// TIA Portal project "lab1" (V15.1)

(* hardware
DEVICE "S7-1200 station_1"  S7-1200 Station
   slot 0: "Rack_0"  S7-1200 Rack  Rack  V1.0
   slot 1: "PLC_1"  CPU 1214C AC/DC/Rly  6ES7 214-1BG40-0XB0  V4.2
*)

// ===== PLC "PLC_1"  CPU 1214C AC/DC/Rly =====

VAR_GLOBAL   // PLC tag table "Default tag table"
   "START_NO" AT %I0.1 : Bool;
   "MOTOR_RADI_NO" AT %I0.2 : Bool;
   "AUTOMATSKI_REZIM_NO" AT %I0.3 : Bool;
   "STOP_NO" AT %I0.5 : Bool;
   "SAFETY_RELE_NC" AT %I0.6 : Bool;
   "ZASTITNI_PREKIDAC_NO" AT %I1.0 : Bool;
   "KONTAKTOR_UKLJUCEN_NO" AT %I1.1 : Bool;
   "ZELENI_LED" AT %Q0.0 : Bool;
   "CRVENI_LED" AT %Q0.1 : Bool;
   "KONTAKTOR_IZLAZ" AT %Q0.2 : Bool;
   "KVAR_ZASTITNI_PREKIDAC" AT %M0.0 : Bool;
   "KVAR_KONTAKTOR" AT %M0.1 : Bool;
   "KVAR_SAFETY_RELE" AT %M0.2 : Bool;
   "STANJE_MOTORA" AT %M0.3 : Bool;
   "Clock_Byte" AT %MB5000 : Byte;
   "Clock_10Hz" AT %M5000.0 : Bool;
   "Clock_5Hz" AT %M5000.1 : Bool;
   "Clock_2.5Hz" AT %M5000.2 : Bool;
   "Clock_2Hz" AT %M5000.3 : Bool;
   "Clock_1.25Hz" AT %M5000.4 : Bool;
   "Clock_1Hz" AT %M5000.5 : Bool;
   "Clock_0.625Hz" AT %M5000.6 : Bool;
   "Clock_0.5Hz" AT %M5000.7 : Bool;
   "ZABRANA" AT %M0.4 : Bool;
   "BLOKADA" AT %M0.5 : Bool;
   "BLOKADA_PROCES_OTPOCEO" AT %M0.6 : Bool;
   "BLOKADA_JEDAN_DVOKLIK_BROJAC_RESET" AT %M0.7 : Bool;
   "BLOKADA_MOD_VREDNOST_NAIZMENICNI_LED" AT %MW2 : Int;
   "BLOKADA_NEUSPESNA" AT %M4.0 : Bool;
   "BLOKADA_POKUSAJ_ISTEKLO_8_SEKUNDI" AT %M4.1 : Bool;
   "ZELENI_LED_UKLJUCEN_1" AT %M4.2 : Bool;
   "CRVENI_LED_UKLJUCEN_1" AT %M4.3 : Bool;
   "CRVENI_LED_UKLJUCEN_2" AT %M4.4 : Bool;
   "CRVENI_LED_UKLJUCEN_3" AT %M4.5 : Bool;
   "ZELENI_LED_UKLJUCEN_2" AT %M4.6 : Bool;
   "CRVENI_LED_UKLJUCEN_4" AT %M4.7 : Bool;
   "CRVENI_LED_UKLJUCEN_5" AT %M5.0 : Bool;
   "DEBLOKADA_PROCES_OTPOCEO" AT %M5.1 : Bool;
   "DEBLOKADA_POKUSAJ_ISTEKLO_6_SEKUNDI" AT %M5.2 : Bool;
   "INKREMENTIRAN_DEBLOKADA_STOP_KLIK_BROJAC" AT %MW6 : Int;
   "DEBLOKADA" AT %M8.0 : Bool;
   "DEBLOKADA_NEUSPESNA" AT %M8.1 : Bool;
   "CRVENI_LED_UKLJUCEN_6" AT %M8.2 : Bool;
   "DEBLOKADA_SUVISNI_KLIKOVI" AT %M8.3 : Bool;
   "BLOKADA_USPESNA_SIGNALIZACIJA_GOTOVA" AT %M8.4 : Bool;
   "DEBLOKADA_SIGNALIZACIJA_USPESNA" AT %M8.5 : Bool;
   "ZELENI_LED_UKLJUCEN_3" AT %M8.6 : Bool;
   "CRVENI_LED_UKLJUCEN_7" AT %M8.7 : Bool;
   "Clock_0.75Hz" AT %M9.0 : Bool;
END_VAR

DATA_BLOCK "OBRADA_KVAROVA_DB"   // DB16
{ S7_Optimized_Access := 'TRUE' }
VERSION : 0.1
// stored: InstanceOfName OBRADA_KVAROVA
"OBRADA_KVAROVA"
BEGIN
END_DATA_BLOCK

DATA_BLOCK "POKRETANJE_I_ZAUSTAVLJANJE_MOTORA_DB"   // DB19
{ S7_Optimized_Access := 'TRUE' }
VERSION : 0.1
// stored: InstanceOfName POKRETANJE_I_ZAUSTAVLJANJE_MOTORA
"POKRETANJE_I_ZAUSTAVLJANJE_MOTORA"
BEGIN
END_DATA_BLOCK

DATA_BLOCK "GENERISANJE_CLOCK_0.75HZ_DB"   // DB20
{ S7_Optimized_Access := 'TRUE' }
VERSION : 0.1
// stored: InstanceOfName GENERISANJE_CLOCK_0.75HZ
"GENERISANJE_CLOCK_0.75HZ"
BEGIN
END_DATA_BLOCK

DATA_BLOCK "UKLJUCIVANJE_I_ISKLJUCIVANJE_LED_LAMPICA_DB"   // DB21
{ S7_Optimized_Access := 'TRUE' }
VERSION : 0.1
// stored: InstanceOfName UKLJUCIVANJE_I_ISKLJUCIVANJE_LED_LAMPICA
"UKLJUCIVANJE_I_ISKLJUCIVANJE_LED_LAMPICA"
BEGIN
END_DATA_BLOCK

DATA_BLOCK "AKTIVACIJA_I_DEAKTIVACIJA_ZABRANE_DB"   // DB22
{ S7_Optimized_Access := 'TRUE' }
VERSION : 0.1
// stored: InstanceOfName AKTIVACIJA_I_DEAKTIVACIJA_ZABRANE
"AKTIVACIJA_I_DEAKTIVACIJA_ZABRANE"
BEGIN
END_DATA_BLOCK

DATA_BLOCK "IMPLEMENTACIJA_BLOKADE_DB"   // DB23
{ S7_Optimized_Access := 'TRUE' }
VERSION : 0.1
// stored: InstanceOfName IMPLEMENTACIJA_BLOKADE
"IMPLEMENTACIJA_BLOKADE"
BEGIN
END_DATA_BLOCK

DATA_BLOCK "BLOKADA_USPESNA_SIGNALIZACIJA_DB"   // DB24
{ S7_Optimized_Access := 'TRUE' }
VERSION : 0.1
// stored: InstanceOfName BLOKADA_USPESNA_SIGNALIZACIJA
"BLOKADA_USPESNA_SIGNALIZACIJA"
BEGIN
END_DATA_BLOCK

DATA_BLOCK "BLOKADA_NEUSPESNA_SIGNALIZACIJA_DB"   // DB25
{ S7_Optimized_Access := 'TRUE' }
VERSION : 0.1
// stored: InstanceOfName BLOKADA_NEUSPESNA_SIGNALIZACIJA
"BLOKADA_NEUSPESNA_SIGNALIZACIJA"
BEGIN
END_DATA_BLOCK

DATA_BLOCK "IMPLEMENTACIJA_DEBLOKADE_DB"   // DB26
{ S7_Optimized_Access := 'TRUE' }
VERSION : 0.1
// stored: InstanceOfName IMPLEMENTACIJA_DEBLOKADE
"IMPLEMENTACIJA_DEBLOKADE"
BEGIN
END_DATA_BLOCK

DATA_BLOCK "DEBLOKADA_USPESNA_SIGNALIZACIJA_DB"   // DB27
{ S7_Optimized_Access := 'TRUE' }
VERSION : 0.1
// stored: InstanceOfName DEBLOKADA_USPESNA_SIGNALIZACIJA
"DEBLOKADA_USPESNA_SIGNALIZACIJA"
BEGIN
END_DATA_BLOCK

DATA_BLOCK "DEBLOKADA_NEUSPESNA_SIGNALIZACIJA_DB"   // DB28
{ S7_Optimized_Access := 'TRUE' }
VERSION : 0.1
// stored: InstanceOfName DEBLOKADA_NEUSPESNA_SIGNALIZACIJA
"DEBLOKADA_NEUSPESNA_SIGNALIZACIJA"
BEGIN
END_DATA_BLOCK

// folder: System blocks/Program resources

DATA_BLOCK "KONTAKTOR_DB"   // DB1
{ S7_Optimized_Access := 'TRUE' }
AUTHOR : Simatic
FAMILY : IEC
NAME : IEC_TMR
VERSION : 1.0
// stored: InstanceOfName IEC_TIMER
"IEC_TIMER"
BEGIN
END_DATA_BLOCK

DATA_BLOCK "BLOKADA_JEDAN_DVOKLIK_TAJMER"   // DB2
{ S7_Optimized_Access := 'TRUE' }
AUTHOR : Simatic
FAMILY : IEC
NAME : IEC_TMR
VERSION : 1.0
// stored: InstanceOfName IEC_TIMER
"IEC_TIMER"
BEGIN
END_DATA_BLOCK

DATA_BLOCK "BLOKADA_NAIZMENICNI_LED_BROJAC"   // DB3
{ S7_Optimized_Access := 'TRUE' }
AUTHOR : Simatic
FAMILY : IEC
NAME : CNTR
VERSION : 1.0
// stored: InstanceOfName IEC_COUNTER
"IEC_COUNTER"
BEGIN
END_DATA_BLOCK

DATA_BLOCK "BLOKADA_SIGNALIZACIJA_LED_TAJMER"   // DB4
{ S7_Optimized_Access := 'TRUE' }
AUTHOR : Simatic
FAMILY : IEC
NAME : IEC_TMR
VERSION : 1.0
// stored: InstanceOfName IEC_TIMER
"IEC_TIMER"
BEGIN
END_DATA_BLOCK

DATA_BLOCK "BLOKADA_JEDAN_DVOKLIK_BROJAC"   // DB5
{ S7_Optimized_Access := 'TRUE' }
AUTHOR : Simatic
FAMILY : IEC
NAME : CNTR
VERSION : 1.0
// stored: InstanceOfName IEC_COUNTER
"IEC_COUNTER"
BEGIN
END_DATA_BLOCK

DATA_BLOCK "BLOKADA_SEKVENCA_TAJMER_DB"   // DB6
{ S7_Optimized_Access := 'TRUE' }
AUTHOR : Simatic
FAMILY : IEC
NAME : IEC_TMR
VERSION : 1.0
// stored: InstanceOfName IEC_TIMER
"IEC_TIMER"
BEGIN
END_DATA_BLOCK

DATA_BLOCK "BLOKADA_NEUSPESNA_TAJMER"   // DB7
{ S7_Optimized_Access := 'TRUE' }
AUTHOR : Simatic
FAMILY : IEC
NAME : IEC_TMR
VERSION : 1.0
// stored: InstanceOfName IEC_TIMER
"IEC_TIMER"
BEGIN
END_DATA_BLOCK

DATA_BLOCK "BLOKADA_SVI_DVOKLICI_BROJAC"   // DB8
{ S7_Optimized_Access := 'TRUE' }
AUTHOR : Simatic
FAMILY : IEC
NAME : CNTR
VERSION : 1.0
// stored: InstanceOfName IEC_COUNTER
"IEC_COUNTER"
BEGIN
END_DATA_BLOCK

DATA_BLOCK "DEBLOKADA_SEKVENCA_TAJMER"   // DB9
{ S7_Optimized_Access := 'TRUE' }
AUTHOR : Simatic
FAMILY : IEC
NAME : IEC_TMR
VERSION : 1.0
// stored: InstanceOfName IEC_TIMER
"IEC_TIMER"
BEGIN
END_DATA_BLOCK

DATA_BLOCK "DEBLOKADA_START_KLIK_BROJAC"   // DB10
{ S7_Optimized_Access := 'TRUE' }
AUTHOR : Simatic
FAMILY : IEC
NAME : CNTR
VERSION : 1.0
// stored: InstanceOfName IEC_COUNTER
"IEC_COUNTER"
BEGIN
END_DATA_BLOCK

DATA_BLOCK "DEBLOKADA_STOP_KLIK_BROJAC"   // DB11
{ S7_Optimized_Access := 'TRUE' }
AUTHOR : Simatic
FAMILY : IEC
NAME : CNTR
VERSION : 1.0
// stored: InstanceOfName IEC_COUNTER
"IEC_COUNTER"
BEGIN
END_DATA_BLOCK

DATA_BLOCK "DEBLOKADA_JEDAN_KLIK_TAJMER"   // DB12
{ S7_Optimized_Access := 'TRUE' }
AUTHOR : Simatic
FAMILY : IEC
NAME : IEC_TMR
VERSION : 1.0
// stored: InstanceOfName IEC_TIMER
"IEC_TIMER"
BEGIN
END_DATA_BLOCK

DATA_BLOCK "DEBLOKADA_NEUSPESNA_TAJMER"   // DB13
{ S7_Optimized_Access := 'TRUE' }
AUTHOR : Simatic
FAMILY : IEC
NAME : IEC_TMR
VERSION : 1.0
// stored: InstanceOfName IEC_TIMER
"IEC_TIMER"
BEGIN
END_DATA_BLOCK

DATA_BLOCK "DEBLOKADA_USPESNA_SIGNALIZACIJA_TAJMER"   // DB15
{ S7_Optimized_Access := 'TRUE' }
AUTHOR : Simatic
FAMILY : IEC
NAME : IEC_TMR
VERSION : 1.0
// stored: InstanceOfName IEC_TIMER
"IEC_TIMER"
BEGIN
END_DATA_BLOCK

DATA_BLOCK "CLOCK_0.75HZ_TAJMER_VREDNOST_0"   // DB17
{ S7_Optimized_Access := 'TRUE' }
AUTHOR : Simatic
FAMILY : IEC
NAME : IEC_TMR
VERSION : 1.0
// stored: InstanceOfName IEC_TIMER
"IEC_TIMER"
BEGIN
END_DATA_BLOCK

DATA_BLOCK "CLOCK_0.75HZ_TAJMER_VREDNOST_1"   // DB18
{ S7_Optimized_Access := 'TRUE' }
AUTHOR : Simatic
FAMILY : IEC
NAME : IEC_TMR
VERSION : 1.0
// stored: InstanceOfName IEC_TIMER
"IEC_TIMER"
BEGIN
END_DATA_BLOCK

DATA_BLOCK "STOP_KLIK_VALIDAN_ZA_BLOKADU"   // DB29
{ S7_Optimized_Access := 'TRUE' }
AUTHOR : Simatic
FAMILY : IEC
NAME : CNTR
VERSION : 1.0
// stored: InstanceOfName IEC_COUNTER
"IEC_COUNTER"
BEGIN
END_DATA_BLOCK

// folder: (top level)

FUNCTION_BLOCK "OBRADA_KVAROVA"   // FB1, LAD
{ S7_Optimized_Access := 'TRUE' }
VERSION : 0.1
BEGIN

REGION Network 1
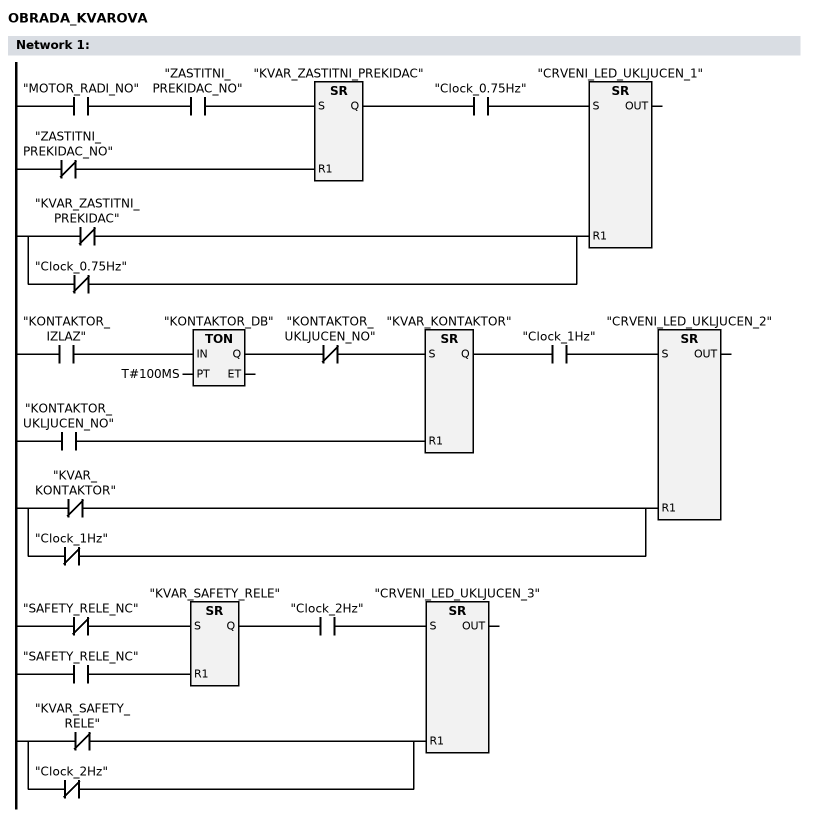
   IF "MOTOR_RADI_NO" AND "ZASTITNI_PREKIDAC_NO" THEN
       "KVAR_ZASTITNI_PREKIDAC" := TRUE;   // SR flip-flop
   END_IF;
   IF NOT "ZASTITNI_PREKIDAC_NO" THEN "KVAR_ZASTITNI_PREKIDAC" := FALSE; END_IF;
   IF "KVAR_ZASTITNI_PREKIDAC" AND "Clock_0.75Hz" THEN
       "CRVENI_LED_UKLJUCEN_1" := TRUE;   // SR flip-flop
   END_IF;
   IF NOT "KVAR_ZASTITNI_PREKIDAC" OR NOT "Clock_0.75Hz" THEN "CRVENI_LED_UKLJUCEN_1" := FALSE; END_IF;
   "KONTAKTOR_DB".TON(IN := "KONTAKTOR_IZLAZ", PT := T#100MS);
   IF "KONTAKTOR_DB".Q AND NOT "KONTAKTOR_UKLJUCEN_NO" THEN
       "KVAR_KONTAKTOR" := TRUE;   // SR flip-flop
   END_IF;
   IF "KONTAKTOR_UKLJUCEN_NO" THEN "KVAR_KONTAKTOR" := FALSE; END_IF;
   IF "KVAR_KONTAKTOR" AND "Clock_1Hz" THEN
       "CRVENI_LED_UKLJUCEN_2" := TRUE;   // SR flip-flop
   END_IF;
   IF NOT "KVAR_KONTAKTOR" OR NOT "Clock_1Hz" THEN "CRVENI_LED_UKLJUCEN_2" := FALSE; END_IF;
   IF NOT "SAFETY_RELE_NC" THEN
       "KVAR_SAFETY_RELE" := TRUE;   // SR flip-flop
   END_IF;
   IF "SAFETY_RELE_NC" THEN "KVAR_SAFETY_RELE" := FALSE; END_IF;
   IF "KVAR_SAFETY_RELE" AND "Clock_2Hz" THEN
       "CRVENI_LED_UKLJUCEN_3" := TRUE;   // SR flip-flop
   END_IF;
   IF NOT "KVAR_SAFETY_RELE" OR NOT "Clock_2Hz" THEN "CRVENI_LED_UKLJUCEN_3" := FALSE; END_IF;
END_REGION
END_FUNCTION_BLOCK

FUNCTION_BLOCK "POKRETANJE_I_ZAUSTAVLJANJE_MOTORA"   // FB2, LAD
{ S7_Optimized_Access := 'TRUE' }
VERSION : 0.1
BEGIN

REGION Network 1
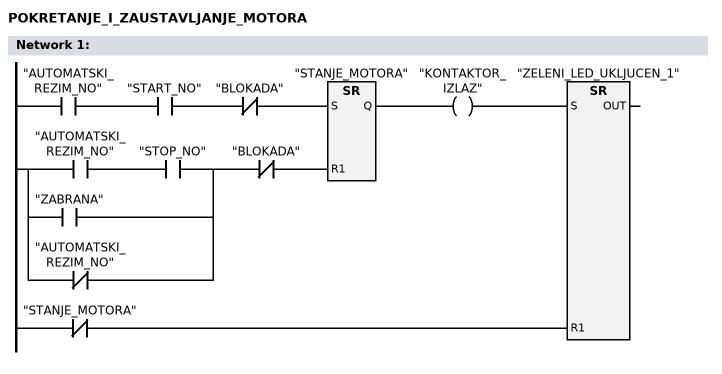
   RUNG wire#powerrail
      Contact( "AUTOMATSKI_REZIM_NO" )
      Contact( "START_NO" )
      I_Contact( "BLOKADA" )
      S_SR(operand := "STANJE_MOTORA", r1 := wire#w2)
      Coil( "KONTAKTOR_IZLAZ" )
      S_SR(operand := "ZELENI_LED_UKLJUCEN_1", r1 := wire#w3)
   END_RUNG
   RUNG wire#powerrail
      Contact( "AUTOMATSKI_REZIM_NO" )
      Contact( "STOP_NO" )
      wire#w1
      I_Contact( "BLOKADA" )
   END_RUNG wire#w2
   RUNG wire#powerrail
      Contact( "ZABRANA" )
   END_RUNG wire#w1
   RUNG wire#powerrail
      I_Contact( "AUTOMATSKI_REZIM_NO" )
   END_RUNG wire#w1
   RUNG wire#powerrail
      I_Contact( "STANJE_MOTORA" )
   END_RUNG wire#w3
   // the same network as SCL:
   IF "AUTOMATSKI_REZIM_NO" AND "START_NO" AND NOT "BLOKADA" THEN
       "STANJE_MOTORA" := TRUE;   // SR flip-flop
   END_IF;
   IF (("AUTOMATSKI_REZIM_NO" AND "STOP_NO") OR "ZABRANA" OR NOT "AUTOMATSKI_REZIM_NO") AND NOT "BLOKADA" THEN
       "STANJE_MOTORA" := FALSE;
   END_IF;
   "KONTAKTOR_IZLAZ" := "STANJE_MOTORA";
   IF "STANJE_MOTORA" THEN
       "ZELENI_LED_UKLJUCEN_1" := TRUE;   // SR flip-flop
   END_IF;
   IF NOT "STANJE_MOTORA" THEN "ZELENI_LED_UKLJUCEN_1" := FALSE; END_IF;
END_REGION
END_FUNCTION_BLOCK

FUNCTION_BLOCK "GENERISANJE_CLOCK_0.75HZ"   // FB3, LAD
{ S7_Optimized_Access := 'TRUE' }
VERSION : 0.1
BEGIN

REGION Network 1
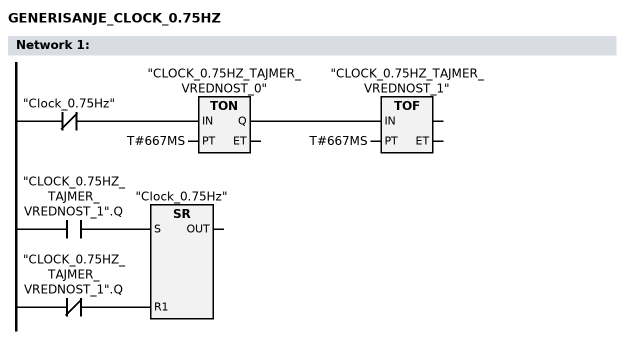
   "CLOCK_0.75HZ_TAJMER_VREDNOST_0".TON(IN := NOT "Clock_0.75Hz", PT := T#667MS);
   "CLOCK_0.75HZ_TAJMER_VREDNOST_1".TOF(IN := "CLOCK_0.75HZ_TAJMER_VREDNOST_0".Q, PT := T#667MS);
   IF "CLOCK_0.75HZ_TAJMER_VREDNOST_1".Q THEN
       "Clock_0.75Hz" := TRUE;   // SR flip-flop
   END_IF;
   IF NOT "CLOCK_0.75HZ_TAJMER_VREDNOST_1".Q THEN "Clock_0.75Hz" := FALSE; END_IF;
END_REGION
END_FUNCTION_BLOCK

FUNCTION_BLOCK "UKLJUCIVANJE_I_ISKLJUCIVANJE_LED_LAMPICA"   // FB4, LAD
{ S7_Optimized_Access := 'TRUE' }
VERSION : 0.1
BEGIN

REGION Network 1
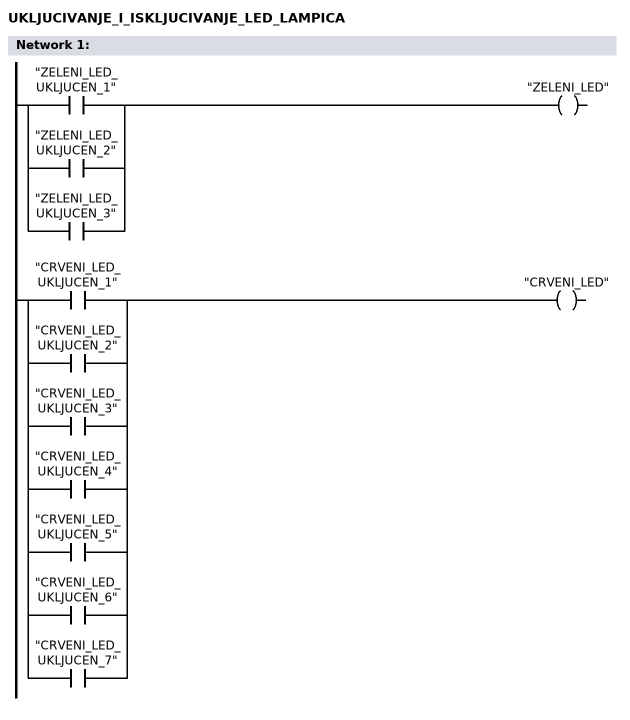
   RUNG wire#powerrail
      Contact( "ZELENI_LED_UKLJUCEN_1" )
      wire#w1
      Coil( "ZELENI_LED" )
   END_RUNG
   RUNG wire#powerrail
      Contact( "ZELENI_LED_UKLJUCEN_2" )
   END_RUNG wire#w1
   RUNG wire#powerrail
      Contact( "ZELENI_LED_UKLJUCEN_3" )
   END_RUNG wire#w1
   RUNG wire#powerrail
      Contact( "CRVENI_LED_UKLJUCEN_1" )
      wire#w2
      Coil( "CRVENI_LED" )
   END_RUNG
   RUNG wire#powerrail
      Contact( "CRVENI_LED_UKLJUCEN_2" )
   END_RUNG wire#w2
   RUNG wire#powerrail
      Contact( "CRVENI_LED_UKLJUCEN_3" )
   END_RUNG wire#w2
   RUNG wire#powerrail
      Contact( "CRVENI_LED_UKLJUCEN_4" )
   END_RUNG wire#w2
   RUNG wire#powerrail
      Contact( "CRVENI_LED_UKLJUCEN_5" )
   END_RUNG wire#w2
   RUNG wire#powerrail
      Contact( "CRVENI_LED_UKLJUCEN_6" )
   END_RUNG wire#w2
   RUNG wire#powerrail
      Contact( "CRVENI_LED_UKLJUCEN_7" )
   END_RUNG wire#w2
   // the same network as SCL:
   "ZELENI_LED" := "ZELENI_LED_UKLJUCEN_1" OR "ZELENI_LED_UKLJUCEN_2" OR "ZELENI_LED_UKLJUCEN_3";
   "CRVENI_LED" := "CRVENI_LED_UKLJUCEN_1" OR "CRVENI_LED_UKLJUCEN_2" OR "CRVENI_LED_UKLJUCEN_3" OR "CRVENI_LED_UKLJUCEN_4" OR "CRVENI_LED_UKLJUCEN_5" OR "CRVENI_LED_UKLJUCEN_6" OR "CRVENI_LED_UKLJUCEN_7";
END_REGION
END_FUNCTION_BLOCK

FUNCTION_BLOCK "AKTIVACIJA_I_DEAKTIVACIJA_ZABRANE"   // FB5, LAD
{ S7_Optimized_Access := 'TRUE' }
VERSION : 0.1
BEGIN

REGION Network 1
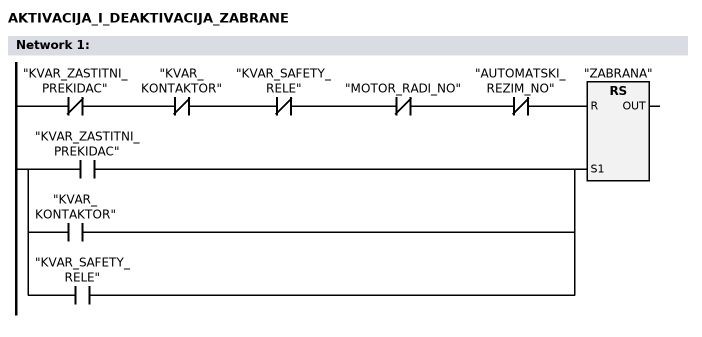
   RUNG wire#powerrail
      I_Contact( "KVAR_ZASTITNI_PREKIDAC" )
      I_Contact( "KVAR_KONTAKTOR" )
      I_Contact( "KVAR_SAFETY_RELE" )
      I_Contact( "MOTOR_RADI_NO" )
      I_Contact( "AUTOMATSKI_REZIM_NO" )
      S_RS(operand := "ZABRANA", s1 := wire#w1)
   END_RUNG
   RUNG wire#powerrail
      Contact( "KVAR_ZASTITNI_PREKIDAC" )
   END_RUNG wire#w1
   RUNG wire#powerrail
      Contact( "KVAR_KONTAKTOR" )
   END_RUNG wire#w1
   RUNG wire#powerrail
      Contact( "KVAR_SAFETY_RELE" )
   END_RUNG wire#w1
   // the same network as SCL:
   IF NOT "KVAR_ZASTITNI_PREKIDAC" AND NOT "KVAR_KONTAKTOR" AND NOT "KVAR_SAFETY_RELE" AND NOT "MOTOR_RADI_NO" AND NOT "AUTOMATSKI_REZIM_NO" THEN
       "ZABRANA" := FALSE;   // RS flip-flop
   END_IF;
   IF "KVAR_ZASTITNI_PREKIDAC" OR "KVAR_KONTAKTOR" OR "KVAR_SAFETY_RELE" THEN "ZABRANA" := TRUE; END_IF;
END_REGION
END_FUNCTION_BLOCK

FUNCTION_BLOCK "IMPLEMENTACIJA_BLOKADE"   // FB6, LAD
{ S7_Optimized_Access := 'TRUE' }
VERSION : 0.1
BEGIN

REGION Network 1
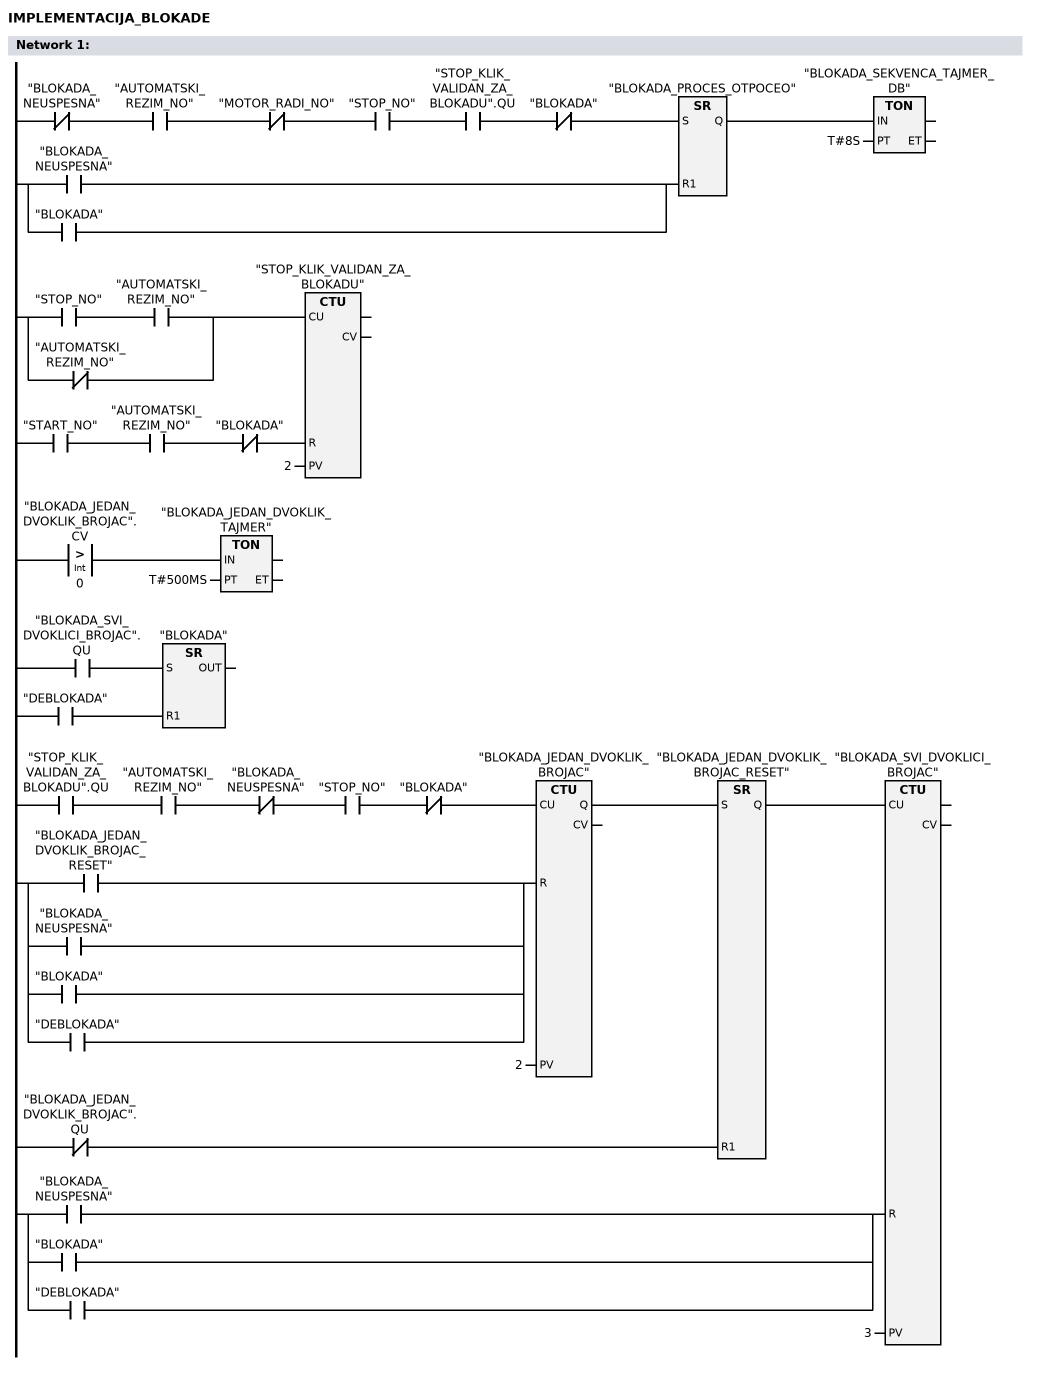
   IF NOT "BLOKADA_NEUSPESNA" AND "AUTOMATSKI_REZIM_NO" AND NOT "MOTOR_RADI_NO" AND "STOP_NO" AND "STOP_KLIK_VALIDAN_ZA_BLOKADU".QU AND NOT "BLOKADA" THEN
       "BLOKADA_PROCES_OTPOCEO" := TRUE;   // SR flip-flop
   END_IF;
   IF "BLOKADA_NEUSPESNA" OR "BLOKADA" THEN "BLOKADA_PROCES_OTPOCEO" := FALSE; END_IF;
   "BLOKADA_SEKVENCA_TAJMER_DB".TON(IN := "BLOKADA_PROCES_OTPOCEO", PT := T#8S);
   "STOP_KLIK_VALIDAN_ZA_BLOKADU".CTU(CU := ("STOP_NO" AND "AUTOMATSKI_REZIM_NO") OR NOT "AUTOMATSKI_REZIM_NO",
                           R := "START_NO" AND "AUTOMATSKI_REZIM_NO" AND NOT "BLOKADA",
                           PV := 2);
   "BLOKADA_JEDAN_DVOKLIK_TAJMER".TON(IN := "BLOKADA_JEDAN_DVOKLIK_BROJAC".CV > 0, PT := T#500MS);
   IF "BLOKADA_SVI_DVOKLICI_BROJAC".QU THEN
       "BLOKADA" := TRUE;   // SR flip-flop
   END_IF;
   IF "DEBLOKADA" THEN "BLOKADA" := FALSE; END_IF;
   "BLOKADA_JEDAN_DVOKLIK_BROJAC".CTU(CU := "STOP_KLIK_VALIDAN_ZA_BLOKADU".QU AND "AUTOMATSKI_REZIM_NO" AND NOT "BLOKADA_NEUSPESNA" AND "STOP_NO" AND NOT "BLOKADA",
                           R := "BLOKADA_JEDAN_DVOKLIK_BROJAC_RESET" OR "BLOKADA_NEUSPESNA" OR "BLOKADA" OR "DEBLOKADA",
                           PV := 2);
   IF "BLOKADA_JEDAN_DVOKLIK_BROJAC".Q THEN
       "BLOKADA_JEDAN_DVOKLIK_BROJAC_RESET" := TRUE;   // SR flip-flop
   END_IF;
   IF NOT "BLOKADA_JEDAN_DVOKLIK_BROJAC".QU THEN "BLOKADA_JEDAN_DVOKLIK_BROJAC_RESET" := FALSE; END_IF;
   "BLOKADA_SVI_DVOKLICI_BROJAC".CTU(CU := "BLOKADA_JEDAN_DVOKLIK_BROJAC_RESET",
                           R := "BLOKADA_NEUSPESNA" OR "BLOKADA" OR "DEBLOKADA",
                           PV := 3);
END_REGION
END_FUNCTION_BLOCK

FUNCTION_BLOCK "BLOKADA_USPESNA_SIGNALIZACIJA"   // FB7, LAD
{ S7_Optimized_Access := 'TRUE' }
VERSION : 0.1
BEGIN

REGION Network 1
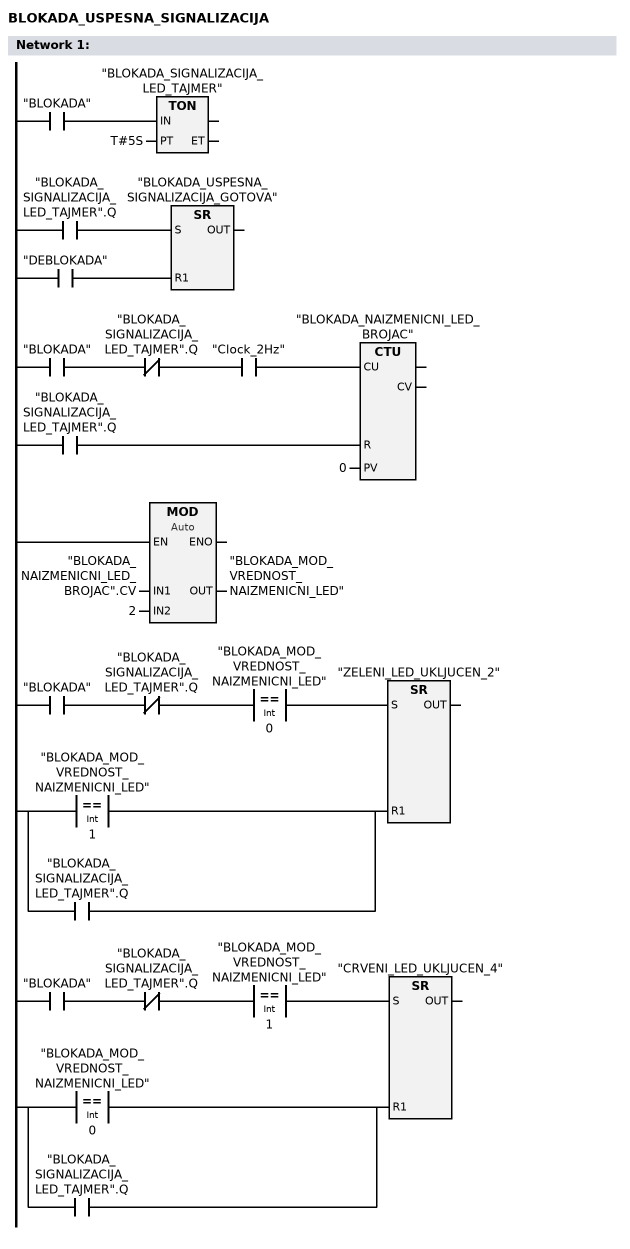
   "BLOKADA_SIGNALIZACIJA_LED_TAJMER".TON(IN := "BLOKADA", PT := T#5S);
   IF "BLOKADA_SIGNALIZACIJA_LED_TAJMER".Q THEN
       "BLOKADA_USPESNA_SIGNALIZACIJA_GOTOVA" := TRUE;   // SR flip-flop
   END_IF;
   IF "DEBLOKADA" THEN "BLOKADA_USPESNA_SIGNALIZACIJA_GOTOVA" := FALSE; END_IF;
   "BLOKADA_NAIZMENICNI_LED_BROJAC".CTU(CU := "BLOKADA" AND NOT "BLOKADA_SIGNALIZACIJA_LED_TAJMER".Q AND "Clock_2Hz",
                           R := "BLOKADA_SIGNALIZACIJA_LED_TAJMER".Q,
                           PV := 0);
   "BLOKADA_MOD_VREDNOST_NAIZMENICNI_LED" := "BLOKADA_NAIZMENICNI_LED_BROJAC".CV MOD 2;
   IF "BLOKADA" AND NOT "BLOKADA_SIGNALIZACIJA_LED_TAJMER".Q AND ("BLOKADA_MOD_VREDNOST_NAIZMENICNI_LED" = 0) THEN
       "ZELENI_LED_UKLJUCEN_2" := TRUE;   // SR flip-flop
   END_IF;
   IF ("BLOKADA_MOD_VREDNOST_NAIZMENICNI_LED" = 1) OR "BLOKADA_SIGNALIZACIJA_LED_TAJMER".Q THEN
       "ZELENI_LED_UKLJUCEN_2" := FALSE;
   END_IF;
   IF "BLOKADA" AND NOT "BLOKADA_SIGNALIZACIJA_LED_TAJMER".Q AND ("BLOKADA_MOD_VREDNOST_NAIZMENICNI_LED" = 1) THEN
       "CRVENI_LED_UKLJUCEN_4" := TRUE;   // SR flip-flop
   END_IF;
   IF ("BLOKADA_MOD_VREDNOST_NAIZMENICNI_LED" = 0) OR "BLOKADA_SIGNALIZACIJA_LED_TAJMER".Q THEN
       "CRVENI_LED_UKLJUCEN_4" := FALSE;
   END_IF;
END_REGION
END_FUNCTION_BLOCK

FUNCTION_BLOCK "BLOKADA_NEUSPESNA_SIGNALIZACIJA"   // FB8, LAD
{ S7_Optimized_Access := 'TRUE' }
VERSION : 0.1
BEGIN

REGION Network 1
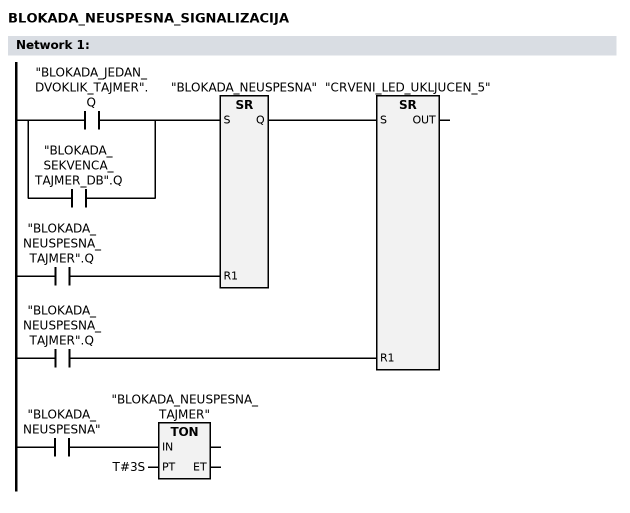
   IF "BLOKADA_JEDAN_DVOKLIK_TAJMER".Q OR "BLOKADA_SEKVENCA_TAJMER_DB".Q THEN
       "BLOKADA_NEUSPESNA" := TRUE;   // SR flip-flop
   END_IF;
   IF "BLOKADA_NEUSPESNA_TAJMER".Q THEN "BLOKADA_NEUSPESNA" := FALSE; END_IF;
   IF "BLOKADA_NEUSPESNA" THEN
       "CRVENI_LED_UKLJUCEN_5" := TRUE;   // SR flip-flop
   END_IF;
   IF "BLOKADA_NEUSPESNA_TAJMER".Q THEN "CRVENI_LED_UKLJUCEN_5" := FALSE; END_IF;
   "BLOKADA_NEUSPESNA_TAJMER".TON(IN := "BLOKADA_NEUSPESNA", PT := T#3S);
END_REGION
END_FUNCTION_BLOCK

FUNCTION_BLOCK "IMPLEMENTACIJA_DEBLOKADE"   // FB9, LAD
{ S7_Optimized_Access := 'TRUE' }
VERSION : 0.1
BEGIN

REGION Network 1
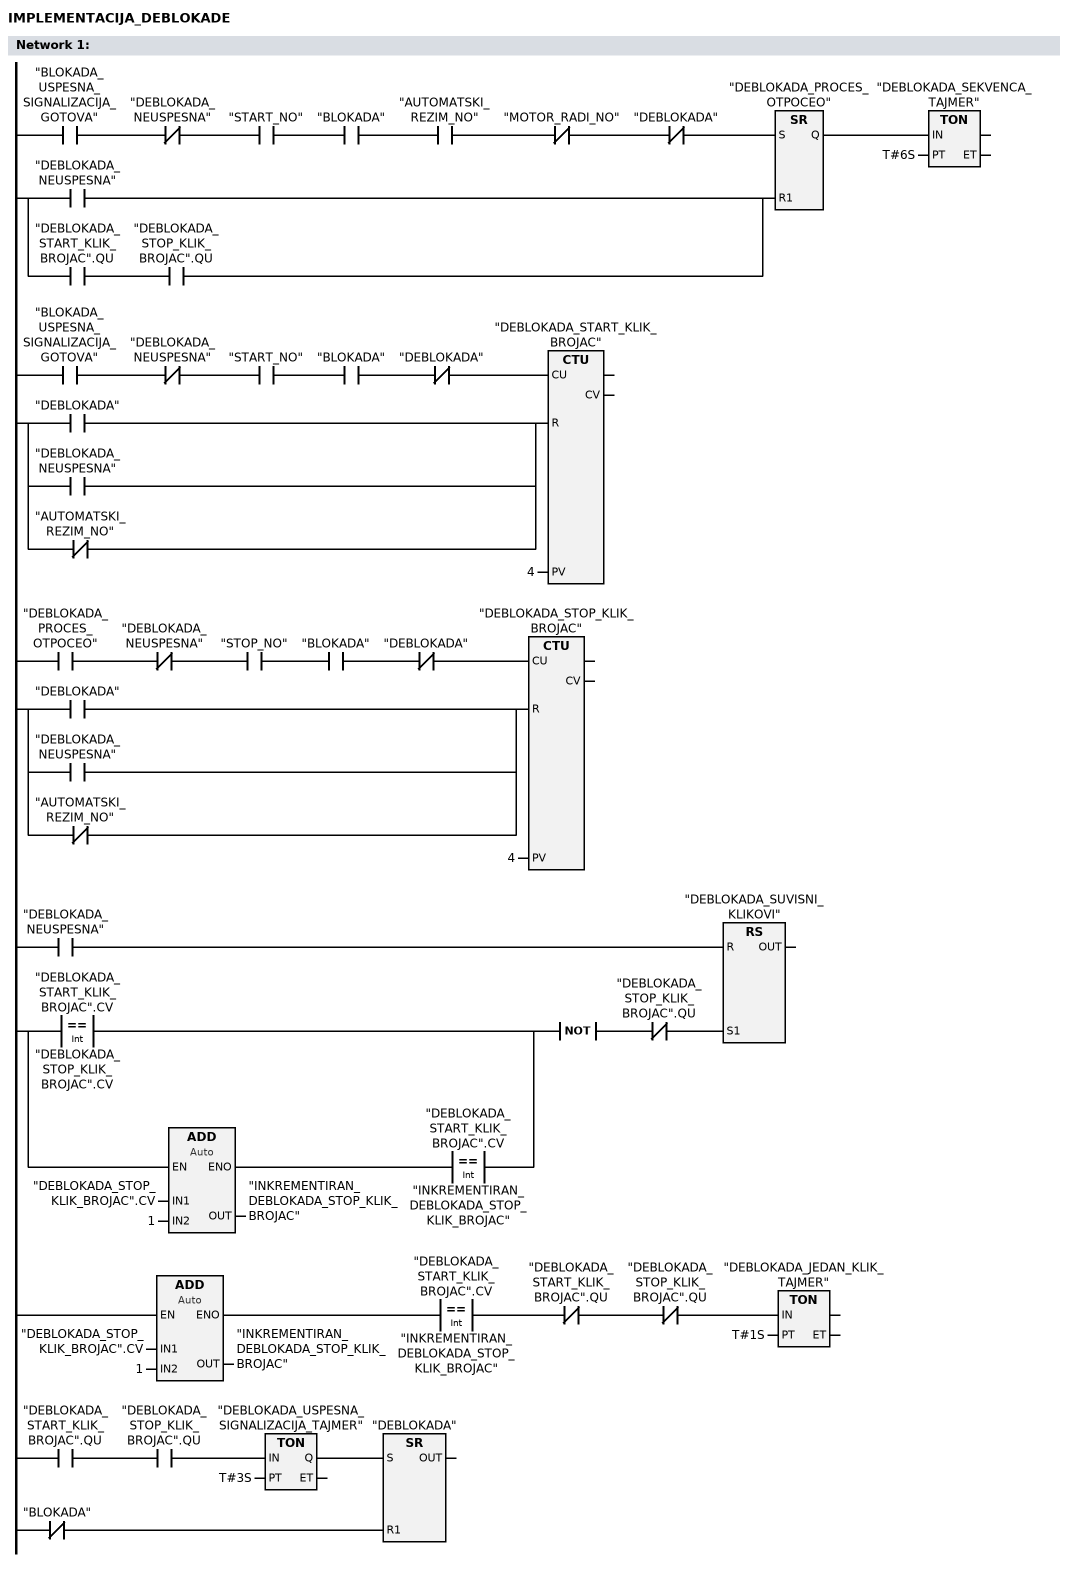
   IF "BLOKADA_USPESNA_SIGNALIZACIJA_GOTOVA" AND NOT "DEBLOKADA_NEUSPESNA" AND "START_NO" AND "BLOKADA" AND "AUTOMATSKI_REZIM_NO" AND NOT "MOTOR_RADI_NO" AND NOT "DEBLOKADA" THEN
       "DEBLOKADA_PROCES_OTPOCEO" := TRUE;   // SR flip-flop
   END_IF;
   IF "DEBLOKADA_NEUSPESNA" OR ("DEBLOKADA_START_KLIK_BROJAC".QU AND "DEBLOKADA_STOP_KLIK_BROJAC".QU) THEN
       "DEBLOKADA_PROCES_OTPOCEO" := FALSE;
   END_IF;
   "DEBLOKADA_SEKVENCA_TAJMER".TON(IN := "DEBLOKADA_PROCES_OTPOCEO", PT := T#6S);
   "DEBLOKADA_START_KLIK_BROJAC".CTU(CU := "BLOKADA_USPESNA_SIGNALIZACIJA_GOTOVA" AND NOT "DEBLOKADA_NEUSPESNA" AND "START_NO" AND "BLOKADA" AND NOT "DEBLOKADA",
                           R := "DEBLOKADA" OR "DEBLOKADA_NEUSPESNA" OR NOT "AUTOMATSKI_REZIM_NO",
                           PV := 4);
   "DEBLOKADA_STOP_KLIK_BROJAC".CTU(CU := "DEBLOKADA_PROCES_OTPOCEO" AND NOT "DEBLOKADA_NEUSPESNA" AND "STOP_NO" AND "BLOKADA" AND NOT "DEBLOKADA",
                           R := "DEBLOKADA" OR "DEBLOKADA_NEUSPESNA" OR NOT "AUTOMATSKI_REZIM_NO",
                           PV := 4);
   "INKREMENTIRAN_DEBLOKADA_STOP_KLIK_BROJAC" := "DEBLOKADA_STOP_KLIK_BROJAC".CV + 1;
   IF "DEBLOKADA_NEUSPESNA" THEN
       "DEBLOKADA_SUVISNI_KLIKOVI" := FALSE;   // RS flip-flop
   END_IF;
   IF NOT (("DEBLOKADA_START_KLIK_BROJAC".CV = "DEBLOKADA_STOP_KLIK_BROJAC".CV) OR ("DEBLOKADA_START_KLIK_BROJAC".CV = "INKREMENTIRAN_DEBLOKADA_STOP_KLIK_BROJAC")) AND NOT "DEBLOKADA_STOP_KLIK_BROJAC".QU THEN
       "DEBLOKADA_SUVISNI_KLIKOVI" := TRUE;
   END_IF;
   "INKREMENTIRAN_DEBLOKADA_STOP_KLIK_BROJAC" := "DEBLOKADA_STOP_KLIK_BROJAC".CV + 1;
   "DEBLOKADA_JEDAN_KLIK_TAJMER".TON(IN := ("DEBLOKADA_START_KLIK_BROJAC".CV = "INKREMENTIRAN_DEBLOKADA_STOP_KLIK_BROJAC") AND NOT "DEBLOKADA_START_KLIK_BROJAC".QU AND NOT "DEBLOKADA_STOP_KLIK_BROJAC".QU,
                           PT := T#1S);
   "DEBLOKADA_USPESNA_SIGNALIZACIJA_TAJMER".TON(IN := "DEBLOKADA_START_KLIK_BROJAC".QU AND "DEBLOKADA_STOP_KLIK_BROJAC".QU,
                           PT := T#3S);
   IF "DEBLOKADA_USPESNA_SIGNALIZACIJA_TAJMER".Q THEN
       "DEBLOKADA" := TRUE;   // SR flip-flop
   END_IF;
   IF NOT "BLOKADA" THEN "DEBLOKADA" := FALSE; END_IF;
END_REGION
END_FUNCTION_BLOCK

FUNCTION_BLOCK "DEBLOKADA_USPESNA_SIGNALIZACIJA"   // FB10, LAD
{ S7_Optimized_Access := 'TRUE' }
VERSION : 0.1
BEGIN

REGION Network 1
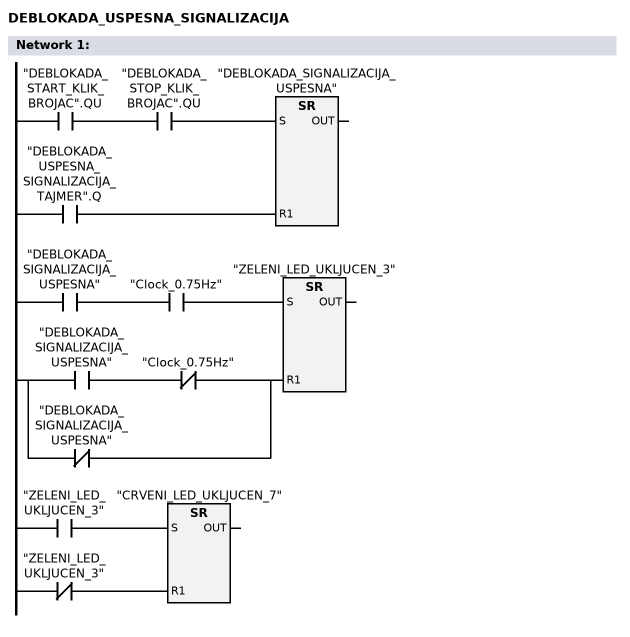
   RUNG wire#powerrail
      Contact( "DEBLOKADA_START_KLIK_BROJAC".QU )
      Contact( "DEBLOKADA_STOP_KLIK_BROJAC".QU )
      S_SR(operand := "DEBLOKADA_SIGNALIZACIJA_USPESNA", r1 := wire#w1)
   END_RUNG
   RUNG wire#powerrail
      Contact( "DEBLOKADA_USPESNA_SIGNALIZACIJA_TAJMER".Q )
   END_RUNG wire#w1
   RUNG wire#powerrail
      Contact( "DEBLOKADA_SIGNALIZACIJA_USPESNA" )
      Contact( "Clock_0.75Hz" )
      S_SR(operand := "ZELENI_LED_UKLJUCEN_3", r1 := wire#w2)
   END_RUNG
   RUNG wire#powerrail
      Contact( "DEBLOKADA_SIGNALIZACIJA_USPESNA" )
      I_Contact( "Clock_0.75Hz" )
   END_RUNG wire#w2
   RUNG wire#powerrail
      I_Contact( "DEBLOKADA_SIGNALIZACIJA_USPESNA" )
   END_RUNG wire#w2
   RUNG wire#powerrail
      Contact( "ZELENI_LED_UKLJUCEN_3" )
      S_SR(operand := "CRVENI_LED_UKLJUCEN_7", r1 := wire#w3)
   END_RUNG
   RUNG wire#powerrail
      I_Contact( "ZELENI_LED_UKLJUCEN_3" )
   END_RUNG wire#w3
   // the same network as SCL:
   IF "DEBLOKADA_START_KLIK_BROJAC".QU AND "DEBLOKADA_STOP_KLIK_BROJAC".QU THEN
       "DEBLOKADA_SIGNALIZACIJA_USPESNA" := TRUE;   // SR flip-flop
   END_IF;
   IF "DEBLOKADA_USPESNA_SIGNALIZACIJA_TAJMER".Q THEN "DEBLOKADA_SIGNALIZACIJA_USPESNA" := FALSE; END_IF;
   IF "DEBLOKADA_SIGNALIZACIJA_USPESNA" AND "Clock_0.75Hz" THEN
       "ZELENI_LED_UKLJUCEN_3" := TRUE;   // SR flip-flop
   END_IF;
   IF ("DEBLOKADA_SIGNALIZACIJA_USPESNA" AND NOT "Clock_0.75Hz") OR NOT "DEBLOKADA_SIGNALIZACIJA_USPESNA" THEN
       "ZELENI_LED_UKLJUCEN_3" := FALSE;
   END_IF;
   IF "ZELENI_LED_UKLJUCEN_3" THEN
       "CRVENI_LED_UKLJUCEN_7" := TRUE;   // SR flip-flop
   END_IF;
   IF NOT "ZELENI_LED_UKLJUCEN_3" THEN "CRVENI_LED_UKLJUCEN_7" := FALSE; END_IF;
END_REGION
END_FUNCTION_BLOCK

FUNCTION_BLOCK "DEBLOKADA_NEUSPESNA_SIGNALIZACIJA"   // FB11, LAD
{ S7_Optimized_Access := 'TRUE' }
VERSION : 0.1
BEGIN

REGION Network 1
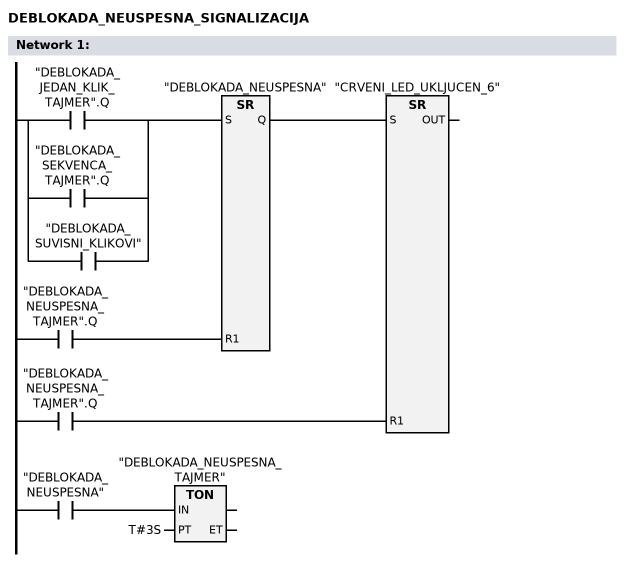
   IF "DEBLOKADA_JEDAN_KLIK_TAJMER".Q OR "DEBLOKADA_SEKVENCA_TAJMER".Q OR "DEBLOKADA_SUVISNI_KLIKOVI" THEN
       "DEBLOKADA_NEUSPESNA" := TRUE;   // SR flip-flop
   END_IF;
   IF "DEBLOKADA_NEUSPESNA_TAJMER".Q THEN "DEBLOKADA_NEUSPESNA" := FALSE; END_IF;
   IF "DEBLOKADA_NEUSPESNA" THEN
       "CRVENI_LED_UKLJUCEN_6" := TRUE;   // SR flip-flop
   END_IF;
   IF "DEBLOKADA_NEUSPESNA_TAJMER".Q THEN "CRVENI_LED_UKLJUCEN_6" := FALSE; END_IF;
   "DEBLOKADA_NEUSPESNA_TAJMER".TON(IN := "DEBLOKADA_NEUSPESNA", PT := T#3S);
END_REGION
END_FUNCTION_BLOCK

ORGANIZATION_BLOCK "Main"   // OB1, LAD, ProgramCycle
TITLE = "Main Program Sweep (Cycle)"
{ S7_Optimized_Access := 'TRUE' }
VERSION : 0.1
   VAR_INPUT
      Initial_Call : Bool;   // Initial call of this OB
      Remanence : Bool;   // =True, if remanent data are available
   END_VAR
BEGIN

REGION Network 1
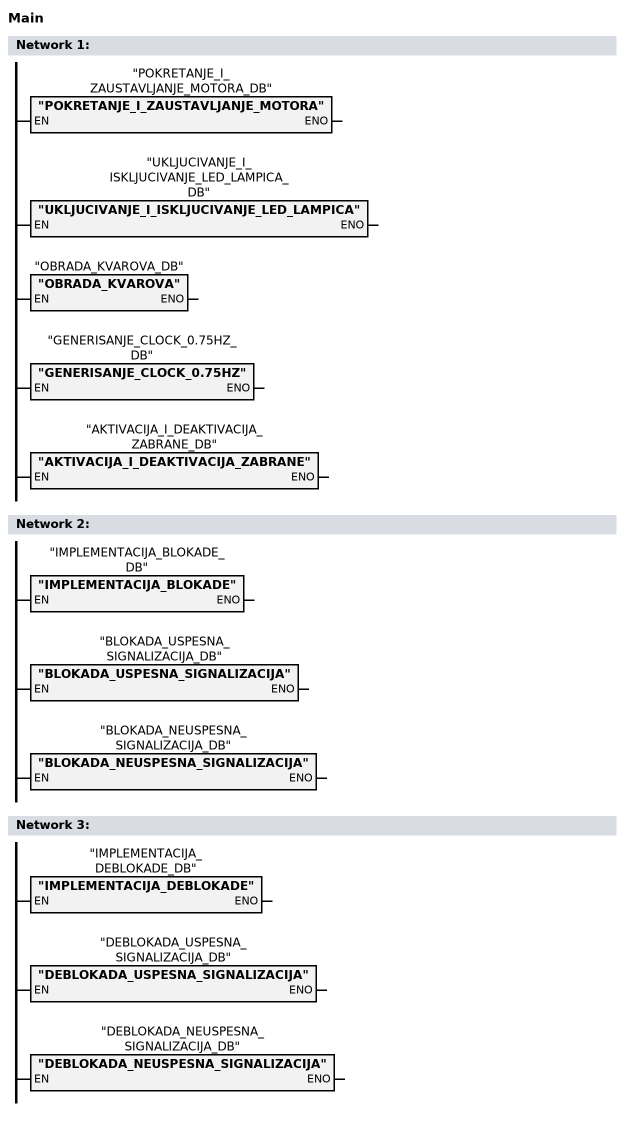
   RUNG wire#powerrail
      "POKRETANJE_I_ZAUSTAVLJANJE_MOTORA_DB"()
   END_RUNG
   RUNG wire#powerrail
      "UKLJUCIVANJE_I_ISKLJUCIVANJE_LED_LAMPICA_DB"()
   END_RUNG
   RUNG wire#powerrail
      "OBRADA_KVAROVA_DB"()
   END_RUNG
   RUNG wire#powerrail
      "GENERISANJE_CLOCK_0.75HZ_DB"()
   END_RUNG
   RUNG wire#powerrail
      "AKTIVACIJA_I_DEAKTIVACIJA_ZABRANE_DB"()
   END_RUNG
   // the same network as SCL:
   "POKRETANJE_I_ZAUSTAVLJANJE_MOTORA_DB"();   // "POKRETANJE_I_ZAUSTAVLJANJE_MOTORA"
   "UKLJUCIVANJE_I_ISKLJUCIVANJE_LED_LAMPICA_DB"();   // "UKLJUCIVANJE_I_ISKLJUCIVANJE_LED_LAMPICA"
   "OBRADA_KVAROVA_DB"();   // "OBRADA_KVAROVA"
   "GENERISANJE_CLOCK_0.75HZ_DB"();   // "GENERISANJE_CLOCK_0.75HZ"
   "AKTIVACIJA_I_DEAKTIVACIJA_ZABRANE_DB"();   // "AKTIVACIJA_I_DEAKTIVACIJA_ZABRANE"
END_REGION

REGION Network 2
   RUNG wire#powerrail
      "IMPLEMENTACIJA_BLOKADE_DB"()
   END_RUNG
   RUNG wire#powerrail
      "BLOKADA_USPESNA_SIGNALIZACIJA_DB"()
   END_RUNG
   RUNG wire#powerrail
      "BLOKADA_NEUSPESNA_SIGNALIZACIJA_DB"()
   END_RUNG
   // the same network as SCL:
   "IMPLEMENTACIJA_BLOKADE_DB"();   // "IMPLEMENTACIJA_BLOKADE"
   "BLOKADA_USPESNA_SIGNALIZACIJA_DB"();   // "BLOKADA_USPESNA_SIGNALIZACIJA"
   "BLOKADA_NEUSPESNA_SIGNALIZACIJA_DB"();   // "BLOKADA_NEUSPESNA_SIGNALIZACIJA"
END_REGION

REGION Network 3
   RUNG wire#powerrail
      "IMPLEMENTACIJA_DEBLOKADE_DB"()
   END_RUNG
   RUNG wire#powerrail
      "DEBLOKADA_USPESNA_SIGNALIZACIJA_DB"()
   END_RUNG
   RUNG wire#powerrail
      "DEBLOKADA_NEUSPESNA_SIGNALIZACIJA_DB"()
   END_RUNG
   // the same network as SCL:
   "IMPLEMENTACIJA_DEBLOKADE_DB"();   // "IMPLEMENTACIJA_DEBLOKADE"
   "DEBLOKADA_USPESNA_SIGNALIZACIJA_DB"();   // "DEBLOKADA_USPESNA_SIGNALIZACIJA"
   "DEBLOKADA_NEUSPESNA_SIGNALIZACIJA_DB"();   // "DEBLOKADA_NEUSPESNA_SIGNALIZACIJA"
END_REGION
END_ORGANIZATION_BLOCK

ORGANIZATION_BLOCK "Startup"   // OB100, LAD, Startup
TITLE = "Complete Restart"
{ S7_Optimized_Access := 'TRUE' }
VERSION : 0.1
   VAR_INPUT
      LostRetentive : Bool;   // True if retentive data are lost
      LostRTC : Bool;   // True if date and time are lost
   END_VAR
BEGIN

REGION Network 1
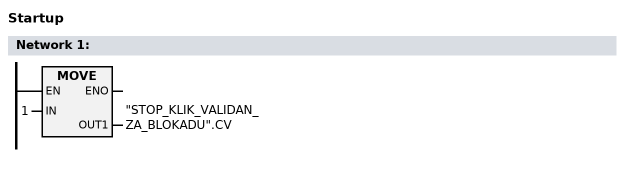
   RUNG wire#powerrail
      Move(in := 1, out1 => "STOP_KLIK_VALIDAN_ZA_BLOKADU".CV)
   END_RUNG
   // the same network as SCL:
   "STOP_KLIK_VALIDAN_ZA_BLOKADU".CV := 1;
END_REGION
END_ORGANIZATION_BLOCK